{attribute 'qualified_only'}
{attribute 'OPC.UA.DA' := '1'}
// Owner-local, bounded publication of the demo's physical CX2030 I/O tree.
// ST_IoChannel.Name is always the exact electrical-list/schematic tag.
VAR_GLOBAL
    Topology : ST_FieldbusTopology;
END_VAR

(* stored: Version 1.1.0.1, ProductVersion 3.1.4024.12
   GVL GVL_PressFieldbus: Id {a3646726-391b-4c93-950c-6c1282fdb93f} *)
